FUNCTION F_counter : INT
VAR_INPUT
	iCounter : INT := 0;
	iCounterStep : INT;
END_VAR
VAR

END_VAR

iCounter := iCounter +iCounterStep;

F_counter := iCounter;

END_FUNCTION

(* stored: Version 1.1.0.1, ProductVersion 3.1.4024.9
   POU F_counter: Id {5a2d1e63-af9a-4b6f-b619-74f720bc8095}, SpecialFunc None *)
